SUBAPPLICATION Ventilsteuerung (* Subapplication Type *)
  (* Standard: 61499-2 *)
  (* Version 1.0, 2023-10-23, franz *)
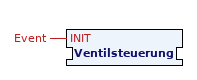
  EVENT_INPUT
    INIT;
  END_EVENT
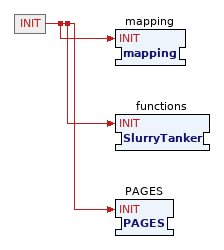
  (* Group Ventilsteuerung: *)
  SUBAPPS
    mapping : mapping; {SET_ATTRIBUTE(GroupName, Ventilsteuerung)}
    functions : SlurryTanker; {SET_ATTRIBUTE(GroupName, Ventilsteuerung)}
    PAGES : PAGES; {SET_ATTRIBUTE(GroupName, Ventilsteuerung)}
  END_SUBAPPS
  EVENT_CONNECTIONS
    INIT TO mapping.INIT;
    INIT TO functions.INIT;
    INIT TO PAGES.INIT;
  END_CONNECTIONS
END_SUBAPPLICATION
